TYPE E_AutomaticMode :
(
	eAuto_reset,
	eAuto_ready,
	eAuto_searchOrder,
	eAuto_noOrder,
	eAuto_approachPosition,
	eAuto_weld
);
END_TYPE

(* stored: Version 1.1.0.1
   DUT E_AutomaticMode: Id {e90f10f9-2537-481f-9180-7040d1d63124} *)
